FUNCTION_BLOCK ABSTRACT SectionEx
VAR_INPUT
	enable : BOOL;
	sectionID : SectionEnum;
END_VAR
VAR_IN_OUT
	bundlesQueue : ARRAY[*] OF Bundle;
	bundlesBypass : ARRAY[*] OF BOOL; //if true, then bypass current bundle
	
	conveyorsArr : ARRAY[*] OF POINTER TO ConveyorSC;
	//in addition to the conveyos array, each section must receive references to the origial conveyors the array elements point to
END_VAR
VAR_OUTPUT
	bundleOut : Bundle; //assigned if there is a bundle to target
	bypass : BOOL; //assigned once the bundle head passes the section (status >= ACTIVE)
END_VAR
VAR_OUTPUT //PackML states + controls
	pmlModeString : STRING;
	pmlStateString : STRING;
	
	stop : BOOL;
	execute : BOOL;
	hold : BOOL;
	reset : BOOL;
	
	ready : BOOL;
	busy : BOOL;
	done : BOOL;
	error : BOOL;
	
	iBundle : INT(0..Consts.maxQueue);
	iPair : INT(0..Consts.maxPairs);
END_VAR
VAR
	pmlState : E_PMLState;
	pmlCommand : E_PMLCommand;
	pmlStateMachine : PML_StateMachine;
	
	pmlModeRequest : E_PMLCustomUnitMode := ePMLCustomUnitMode_Production;
	pmlMode : E_PMLCustomUnitMode;
	pmlModeManager : PML_UnitModeManager;
END_VAR
VAR
	currentBundle : REFERENCE TO Bundle;
	currentBypass : REFERENCE TO BOOL;
	
	loaded : BOOL;
	loadedMaterials : ARRAY[Surface.TOP..Surface.BOTTOM_RIGHT] OF STRING;
	
	entryRefPos : (*REFERENCE TO*) REAL;
	exitRefPos : (*REFERENCE TO*) REAL;
	
	requestedConveyorMode : ConveyorMode;
	
	nextSection : POINTER TO SectionEx;
	prevSection : POINTER TO SectionEx;
	
	occupied : BOOL; //may need to move this to Hardware GVL since this is a sensor
	
	status : SectionTask; //section status
END_VAR
VAR_STAT CONSTANT
	INCLUSIVE : INT := 0;
	EXCLUSIVE : INT := 1;
	COMPLETE : INT := 1030;
	
	suctionReleaseDelay : TIME := T#1000MS;
END_VAR

currentBundle REF= bundlesQueue[iBundle];
currentBypass REF= bundlesBypass[iBundle];
bypass := currentBypass;

ready := status = 0;
busy := status > 0;
done := done;
error := error;

blocks();

runPmlStates();

METHOD PROTECTED blocks : BOOL
pmlModeManager(
	bExecute:= NOT pmlModeManager.bExecute, 
	eModeCommand:= pmlModeRequest, 
	eState:= pmlState, 
	eModeStatus=> pmlMode, 
	sModeStatus=> pmlModeString, 
	bDone=> , 
	bError=> , 
	nErrorId=> );

pmlStateMachine(
	eMode:= pmlMode, 
	eCommand:= pmlCommand, 
	stSubUnitInfoRef:= , 
	stOptions:= , 
	eState=> pmlState, 
	sState=> pmlStateString, 
	bError=> , 
	nErrorID=> );
END_METHOD

METHOD PROTECTED ABSTRACT callLocalModules : BOOL
END_METHOD

METHOD connectTo : BOOL
VAR_INPUT
	connectedSection : POINTER TO SectionEx;
END_VAR
nextSection := connectedSection;

IF connectedSection <> 0 THEN
	connectedSection^.prevSection := THIS;
END_IF
END_METHOD

METHOD PROTECTED directionCheckAndSet : BOOL
VAR_INPUT
	conveyorRef : REAL;
	target : REAL;
END_VAR
//returns true conveyorRef is in range of target
IF InRange(conveyorRef - Consts.precisionTolerance, conveyorRef + Consts.precisionTolerance, target, EXCLUSIVE) THEN
	directionCheckAndSet := TRUE;
	
ELSIF conveyorRef > target THEN
	pConveyorMode := ConveyorMode.BACKWARD;
	
ELSIF conveyorRef < target THEN
	pConveyorMode := ConveyorMode.FORWARD;
	
END_IF
END_METHOD

METHOD PROTECTED ABSTRACT load : BOOL
VAR_INPUT
	pairIndex : INT;
END_VAR
VAR_OUTPUT
	error : BOOL;
END_VAR
(*
loading takes place while the section is NOT active
materials are loaded for the next incoming bundle, not the current bundle - may differ for each section
*)
END_METHOD

METHOD PROTECTED ABSTRACT maintenance : BOOL
VAR_INPUT
END_VAR
END_METHOD

PROPERTY PROTECTED pConveyorMode : ConveyorMode
GET
pConveyorMode := requestedConveyorMode;
END_GET
SET
VAR
	i : DINT;
END_VAR
requestedConveyorMode := pConveyorMode;

FOR i:=LOWER_BOUND(conveyorsArr, 1) TO UPPER_BOUND(conveyorsArr, 1) BY 1 DO
	
	CASE status OF
		SectionTask.ALIGNING, -100:
			//all conveyors requested to same mode
			conveyorsArr[i]^.setRequest(requestedConveyorMode);
			
		SectionTask.ACTIVE, SectionTask.CLEARING:
			//once previous bundle catches up, the conveyor that bundle sits on must be linked to this section
			//a conveyor control module will handle linking
			
			IF conveyorsArr[i]^.IsOccupied THEN //follow this section's request
				conveyorsArr[i]^.setRequest(requestedConveyorMode);
				
			ELSE //catch up succeeding bundle (FOLLOW PREVIOUS SECTION)
				IF prevSection <> 0 THEN
					conveyorsArr[i]^.setRequest( prevSection^.pConveyorMode );
				END_IF
			END_IF
	END_CASE	
	
END_FOR
END_SET
END_PROPERTY

METHOD PROTECTED ABSTRACT process : BOOL
VAR_INPUT
	auto : BOOL;
END_VAR
VAR_OUTPUT
	error : BOOL;
END_VAR
(*
this method is implemented by each section according to their material packaging steps
*)
END_METHOD

METHOD PROTECTED ABSTRACT ps_AbortCondition : BOOL
VAR_INPUT
END_VAR
END_METHOD

METHOD PROTECTED ABSTRACT ps_Aborted : BOOL
VAR_INPUT
END_VAR
END_METHOD

METHOD PROTECTED ABSTRACT ps_Aborting : BOOL
VAR_INPUT
END_VAR
END_METHOD

METHOD PROTECTED ABSTRACT ps_Clearing : BOOL
VAR_INPUT
END_VAR
END_METHOD

METHOD PROTECTED ABSTRACT ps_Complete : BOOL
VAR_INPUT
END_VAR
END_METHOD

METHOD PROTECTED ABSTRACT ps_Completing : BOOL
VAR_INPUT
END_VAR
END_METHOD

METHOD PROTECTED ps_Execute : BOOL
VAR_INPUT
END_VAR
VAR_OUTPUT
	error : BOOL;
END_VAR
CASE pmlMode OF
	0: //invalid mode
	ePMLCustomUnitMode_Production:		ps_Execute := runSectionTasks(auto := TRUE);
	ePMLCustomUnitMode_Maintenance:		maintenance();
	ePMLCustomUnitMode_Manual:			//
	ePMLCustomUnitMode_SemiAuto:		ps_Execute := runSectionTasks(auto := FALSE);
END_CASE
END_METHOD

METHOD PROTECTED ABSTRACT ps_Held : BOOL
VAR_INPUT
END_VAR
END_METHOD

METHOD PROTECTED ABSTRACT ps_HoldCondition : BOOL
VAR_INPUT
END_VAR
END_METHOD

METHOD PROTECTED ABSTRACT ps_Holding : BOOL
VAR_INPUT
END_VAR
END_METHOD

METHOD PROTECTED (*ABSTRACT*) ps_Idle : BOOL
VAR_INPUT
END_VAR
(*
IF BundleIsValid(currentBundle) THEN
	ps_Idle := TRUE;
	done := FALSE;
END_IF
*)

ps_Idle := TRUE; (*start section input*)
END_METHOD

METHOD PROTECTED ABSTRACT ps_Resetting : BOOL
VAR_INPUT
END_VAR
END_METHOD

METHOD PROTECTED ABSTRACT ps_Starting : BOOL
VAR_INPUT
END_VAR
END_METHOD

METHOD PROTECTED ABSTRACT ps_StopCondition : BOOL
VAR_INPUT
END_VAR
END_METHOD

METHOD PROTECTED ABSTRACT ps_Stopped : BOOL
VAR_INPUT
END_VAR
END_METHOD

METHOD PROTECTED ABSTRACT ps_Stopping : BOOL
VAR_INPUT
END_VAR
END_METHOD

METHOD PROTECTED ABSTRACT ps_SuspendCondition : BOOL
VAR_INPUT
END_VAR
END_METHOD

METHOD PROTECTED ABSTRACT ps_Suspended : BOOL
VAR_INPUT
END_VAR
END_METHOD

METHOD PROTECTED ABSTRACT ps_Suspending : BOOL
VAR_INPUT
END_VAR
END_METHOD

METHOD PROTECTED ABSTRACT ps_Unholding : BOOL
VAR_INPUT
END_VAR
END_METHOD

METHOD PROTECTED ABSTRACT ps_Unsuspending : BOOL
VAR_INPUT
END_VAR
END_METHOD

PROPERTY PROTECTED pStatus : SectionTask
GET
pStatus := status;
END_GET
SET
status := pStatus;
END_SET
END_PROPERTY

METHOD PROTECTED runPmlStates : BOOL
(*
PackML
	state machine for packaging applications - see Tc3_PackML_V2 library on InfoSys
	
	final states - wait for an input or condition and command to new state
	intermediate states - complete a task and call pmlStateMachine.M_StateComplete() to advance to next state
	
the following states currently use the same logic (albeit in different methods), implementation may change later
	ps_Stopping() and ps_Aborting()
	ps_Resetting() and ps_Clearing()
	
STOP - controlled stop **with intent to shutdown or vacate for extended time** induced by operator/HMI - otherwise use HOLD
ABORT - emergency stop due to machine errors


HOLD - minor local issues
SUSPEND - external issues

EXECUTE - major control logic
	different modes may require different tasks
	create methods as required for different modes, then call the correct method in ps_Completing()
	can be commanded to STOP, ABORT, HOLD, or SUSPEND at any point
COMPLETING - process complete, move product out of system and finish transition to COMPLETED

the implementation below can be copied to all POUs that use a PackML state machine
the individual ps_< > methods need to be implemented for the specific application
*)


IF ps_AbortCondition() THEN //abort condition
	pmlCommand := ePMLCommand_Abort;
ELSIF ps_StopCondition() THEN //stop condition
	pmlCommand := ePMLCommand_Stop;
END_IF

CASE pmlState OF
	0 (*ePMLState_Undefined*): //default state on startup
		pmlCommand := ePMLCommand_Stop;
		
	ePMLState_Stopping:
		IF ps_Stopping() THEN
			pmlStateMachine.M_StateComplete();
		END_IF
		
	ePMLState_Stopped:
		IF ps_Stopped() THEN
			pmlCommand := ePMLCommand_Reset;
		END_IF
	
    ePMLState_Resetting:
		IF ps_Resetting() THEN
			pmlStateMachine.M_StateComplete();
		END_IF
		
	ePMLState_Idle:
		IF ps_Idle() THEN
			pmlCommand := ePMLCommand_Start;
		END_IF		
	
	ePMLState_Starting:
		IF ps_Starting() THEN
			pmlStateMachine.M_StateComplete();
		END_IF
	
	ePMLState_Execute: //check the conditions in order of their priority, currently HOLD has the highest priority
		IF ps_HoldCondition() THEN
			pmlCommand := ePMLCommand_Hold;
			
		ELSIF ps_SuspendCondition() THEN
			pmlCommand := ePMLCommand_Suspend;			
		
		ELSIF ps_Execute(error => error) THEN //ps_Execute.error => THIS^.error
			pmlStateMachine.M_StateComplete();
			pmlCommand := ePMLCommand_Complete;
		END_IF
		
	ePMLState_Completing:
		IF ps_Completing() THEN
			pmlStateMachine.M_StateComplete();
		END_IF
	
	ePMLState_Complete:
		IF ps_Complete() THEN
			pmlCommand := ePMLCommand_Reset;
		END_IF
	
	ePMLState_Holding:
		IF ps_Holding() THEN
			pmlStateMachine.M_StateComplete();
		END_IF
	
	ePMLState_Held:
		IF NOT hold THEN
			pmlCommand := ePMLCommand_Unhold;
		END_IF
	
	ePMLState_Unholding:
		IF ps_Unholding() THEN
			pmlStateMachine.M_StateComplete(); //release all pause commands and IO
		END_IF
		
	ePMLState_Suspending: //based on next section conditions
		IF ps_Suspending() THEN
			pmlStateMachine.M_StateComplete();
		END_IF
		
	ePMLState_Suspended: //based on next section conditions
		IF ps_Suspended() THEN
			pmlCommand := ePMLCommand_Unsuspend;
		END_IF
	
	ePMLState_Unsuspending: //based on next section conditions
		IF ps_Unsuspending() THEN
			pmlStateMachine.M_StateComplete();
		END_IF
	
	ePMLState_Aborting:
		IF ps_Aborting() THEN
			pmlStateMachine.M_StateComplete();
		END_IF
	
	ePMLState_Aborted:
		IF ps_Aborted() THEN
			pmlCommand := ePMLCommand_Clear;
		END_IF
	
	ePMLState_Clearing:
		IF ps_Clearing() THEN
			pmlStateMachine.M_StateComplete();
		END_IF
	
END_CASE
END_METHOD

METHOD PROTECTED FINAL runSectionTasks : BOOL
VAR_INPUT
	auto : BOOL;
END_VAR
VAR
	error : BOOL;
END_VAR
CASE status OF
	SectionTask.IDLE:
		IF BundleIsValid(currentBundle) THEN			
			status := SectionTask.ALIGNING;
			done := FALSE;
		END_IF
	
	SectionTask.ALIGNING:		
		pConveyorMode := ConveyorMode.FORWARD;
		
		IF 
			occupied AND
			nextSection <> 0 AND
			nextSection^.pConveyorMode = ConveyorMode.BACKWARD
		THEN //section occupied by next section backing up into this section
			status := -100;
			
		ELSIF occupied THEN //section occupied by correct bundle
			//stop and zero the conveyors
			IF NOT auto OR_ELSE execute THEN
				status := SectionTask.ACTIVE;
			END_IF
		END_IF
		
	SectionTask.ACTIVE:
		bundleOut := currentBundle;
		
		IF NOT enable THEN
			iPair := 0;
			status := SectionTask.CLEARING;
			
		ELSIF NOT usesProcess() THEN //bundle does not use this section's processes
			iPair := 0;
			status := SectionTask.CLEARING;
		
		ELSIF currentBypass (*AND_THEN discharge()*) THEN //bundle failed in previous section, discharge this section's materials
			IF unload() THEN
				iPair := 0;
				status := SectionTask.CLEARING;
			END_IF
			
		ELSIF process(auto := auto, error => error) THEN //bundle recipe completed normally
			IF NOT auto OR_ELSE execute THEN
				iPair := 0;
				status := SectionTask.CLEARING;
			END_IF			
		END_IF
		
	SectionTask.CLEARING:
		bundleOut := currentBundle;
		pConveyorMode := ConveyorMode.FORWARD;
		
		IF exitRefPos >= currentBundle.length AND NOT occupied THEN //rear of bundle has cleared the area
			status := SectionTask.COMPLETE;
		END_IF
		
	SectionTask.COMPLETE:	
		iBundle := iBundle + 1;
		//bundleOut := GVL.nullBundle;
		MEMSET(ADR(bundleOut), 0, SIZEOF(bundleOut));
		
		status := SectionTask.IDLE;
		
		runSectionTasks := TRUE;
		
	-100: //previously completed bundle reversed into this section		
		pConveyorMode := ConveyorMode.FORWARD;
		
		IF NOT occupied THEN
			status := SectionTask.ALIGNING;
		END_IF
		
END_CASE
END_METHOD

METHOD shiftIterator : BOOL
VAR
	i : INT;
END_VAR
//2023-10-24 - array of pointers replaced with iterator for MAIN's queue passed by pointer
iBundle := iBundle - 1;
END_METHOD

METHOD PROTECTED ABSTRACT unload : BOOL
VAR_INPUT
END_VAR
(*
unload, unstage, etc
*)
END_METHOD

METHOD PROTECTED ABSTRACT usesProcess : BOOL
(*
this method determines if a bundle uses materials that this section provides
if a bundle does not use this section's process, then it can be skipped
*)
END_METHOD

END_FUNCTION_BLOCK

(* stored: Version 1.1.0.1, ProductVersion 3.1.4024.11
   POU SectionEx: Id {553a7cf7-8736-4fc0-93d1-2ae972262b14}, SpecialFunc None
   Folder Abstract: Id {931032f8-8fbc-437e-9feb-8dfcf4d8fa11}
   Folder PML Conditions: Id {8f6247d2-5ca2-410c-b633-82ec4b58b07b}
   Folder PML States: Id {06e2f1cf-cccc-459b-a09f-1383a082a445}
   Folder Properties: Id {35099ffa-f285-4e22-8f2e-31de1316393c}
   Method blocks: Id {ed2226fe-fd00-49fe-b482-5d0d616dd13b}
   Method callLocalModules: Id {01231dfd-d7d7-43f6-abd5-1b692bab6a1f}
   Method connectTo: Id {91d63988-c603-4003-a46a-ea71ce206f50}
   Method directionCheckAndSet: Id {e472cb3d-3b10-43cb-be34-a868e55e86de}
   Method load: Id {f29da0bd-18e9-4eca-8ea7-a82a57710347}
   Method maintenance: Id {82cfe381-4627-47b2-becb-4530cc701c9e}
   Property pConveyorMode: Id {97786c27-ba47-43a5-9b90-47ff6f5d538e}
   Get Get: Id {0ba095f3-28cd-449d-a6ee-3c87c3d0580a}
   Set Set: Id {af1867f9-e8bf-4840-a3e8-76c799395c42}
   Method process: Id {d318af18-2aae-4a8a-9d12-4aa1944ee865}
   Method ps_AbortCondition: Id {ea0e69dc-628b-404a-acfd-eb96c20b5c8b}
   Method ps_Aborted: Id {fd49a85e-d9c2-4872-999c-4e48c3f35296}
   Method ps_Aborting: Id {8970a2ca-c21c-49d9-911e-491db2e7f876}
   Method ps_Clearing: Id {3fe44078-6a1b-4682-a996-b699c18aee67}
   Method ps_Complete: Id {7833c15a-3310-48e7-8e31-e7e76e3a7760}
   Method ps_Completing: Id {38fedc81-0bce-4ee0-9445-9aadde8a30b1}
   Method ps_Execute: Id {73635fe5-de92-40d6-ba2e-8b3bfdfdbb4e}
   Method ps_Held: Id {97712eef-0a76-4f44-b2a5-7edb9768c1c5}
   Method ps_HoldCondition: Id {18584675-3920-466d-95ca-bc68955d5f21}
   Method ps_Holding: Id {ae1a5d1d-c425-41ab-be42-ac322799fb37}
   Method ps_Idle: Id {ff5dce02-ada7-431d-9ee9-3e17c3a65b4e}
   Method ps_Resetting: Id {cb59b9e4-db36-4a6b-b9fd-e8381e0607d8}
   Method ps_Starting: Id {e89dce85-4a66-44ea-857c-1f5cdfba177a}
   Method ps_StopCondition: Id {a23289dd-9264-41ec-8cf7-f6c6d2f4f445}
   Method ps_Stopped: Id {8e007499-8af0-4da7-be9e-f073186adcc7}
   Method ps_Stopping: Id {1dcebf3c-702f-49e3-8dfe-b35094ec6ccc}
   Method ps_SuspendCondition: Id {fc9d4281-9a99-493c-9484-446186deee9d}
   Method ps_Suspended: Id {505c98ae-539c-49e2-a739-19c90e70899f}
   Method ps_Suspending: Id {cced8904-3605-41d0-8646-a0d5e2e475a7}
   Method ps_Unholding: Id {d1211bb0-9bf2-475e-9bc3-fc66e3405f66}
   Method ps_Unsuspending: Id {177b454f-a063-4ea7-a664-efbf79a9bb04}
   Property pStatus: Id {2fc2840f-258c-4643-bc3e-979cfdbf23f2}
   Get Get: Id {b7542eca-dbd5-4cb3-9aab-eccd028bb0c7}
   Set Set: Id {82f7bd0c-e305-45fe-8dbc-8fb426ee0813}
   Method runPmlStates: Id {cc8dcd6f-b841-4037-adba-e94e1c4ef5d7}
   Method runSectionTasks: Id {ff600a76-8305-47bd-9f4f-604426e1af1d}
   Method shiftIterator: Id {2b1c8dba-7a66-41d7-be54-23459718f73e}
   Method unload: Id {264daea0-fc50-4810-8136-0464ba4deabe}
   Method usesProcess: Id {c1b6c909-9917-4b95-9231-7fe23c878d88} *)
